// TIA Portal project "Project9" (V17)

(* hardware
DEVICE "S7-1200 station_1"  S7-1200 Station
   slot 0: "Rack_0"  S7-1200 Rack  Rack  V1.0
   slot 1: "PLC_1"  CPU 1214C AC/DC/Rly  6ES7 214-1BG40-0XB0  V4.2
*)

// ===== PLC "PLC_1"  CPU 1214C AC/DC/Rly =====

VAR_GLOBAL   // PLC tag table "Default tag table"
   "pb1" AT %M0.0 : Bool;
   "pb2" AT %M0.1 : Bool;
   "pb3" AT %M0.2 : Bool;
   "pb4" AT %M0.3 : Bool;
   "Tag_1" AT %MW100 : Int;
   "Tag_2" AT %MW102 : Int;
   "Tag_3" AT %MW104 : Int;
   "Tag_4" AT %MD200 : Real;
   "Tag_5" AT %MD204 : Real;
   "Tag_6" AT %MD208 : Real;
   "Tag_7" AT %MW106 : Int;
   "Tag_8" AT %MW108 : Int;
END_VAR

ORGANIZATION_BLOCK "Main"   // OB1, LAD, ProgramCycle
TITLE = "Main Program Sweep (Cycle)"
{ S7_Optimized_Access := 'TRUE' }
VERSION : 0.1
   VAR_INPUT
      Initial_Call : Bool;   // Initial call of this OB
      Remanence : Bool;   // =True, if remanent data are available
   END_VAR
BEGIN

REGION Network 1
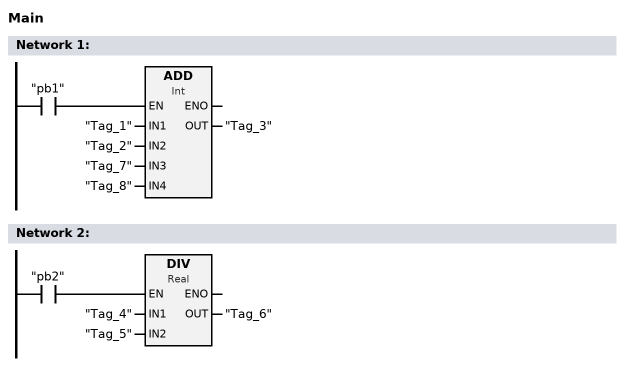
   RUNG wire#powerrail
      Contact( "pb1" )
      { S7_Templates := "SrcType := Int" } Add(in1 := "Tag_1", in2 := "Tag_2", in3 := "Tag_7", in4 := "Tag_8", out => "Tag_3")
   END_RUNG
   // the same network as SCL:
   IF "pb1" THEN "Tag_3" := "Tag_1" + "Tag_2" + "Tag_7" + "Tag_8"; END_IF;
END_REGION

REGION Network 2
   RUNG wire#powerrail
      Contact( "pb2" )
      { S7_Templates := "SrcType := Real" } Div(in1 := "Tag_4", in2 := "Tag_5", out => "Tag_6")
   END_RUNG
   // the same network as SCL:
   IF "pb2" THEN "Tag_6" := "Tag_4" / "Tag_5"; END_IF;
END_REGION
END_ORGANIZATION_BLOCK